TYPE ST_Zustand_Netze_Anford :
STRUCT
	Kaltwasser		: ST_Zustand_Netz_Anford;
	Warmwasser		: ST_Zustand_Netz_Anford;
	Heisswasser		: ST_Zustand_Netz_Anford;
END_STRUCT
END_TYPE

(* stored: Version 1.1.0.1, ProductVersion 3.1.4024.9
   DUT ST_Zustand_Netze_Anford: Id {420df46a-5ed2-4a96-a7aa-e28fe232d658} *)
